TYPE HMIRFIDStatusInterface :
STRUCT
	PermissionHardware	:	BOOL;
	PartPresent	:	BOOL;
	ErrorActive	:	BOOL;
	FMReading	:	BOOL;
	FMWritting	:	BOOL;
END_STRUCT
END_TYPE

(* stored: Version 1.1.0.1
   DUT HMIRFIDStatusInterface: Id {507d6932-9e4b-42eb-9a2d-e47e72ddcb94} *)
